Yaskawa INFORM job: OK_R2_O242(-90,180)OKKR.JBI

/JOB
//NAME OK_R2_O242(-90,180)OKKR
///FOLDERNAME X4
//POS
///NPOS 123,123,123,4,0,0
///TOOL 0
///POSTYPE PULSE
///PULSE
C00000=1085,-105763,-105592,1367,57789,-79187
C00001=48587,-61870,-56373,37554,57186,-71211
C00002=109319,-98863,-81663,-17130,36799,-47258
C00003=110499,-70978,-76585,-14581,28064,-55521
C00004=114923,11399,-23396,-32739,57115,-42289
C00005=116623,27529,-9023,-35345,61036,-36673
C00006=106531,29443,-6029,-23966,54360,-54184
C00007=107072,29107,-4870,-24608,53702,-53789
C00008=107072,28853,-4001,-24811,53095,-53633
C00009=107072,28916,-4224,-24758,53250,-53673
C00010=107722,30543,-2610,-25264,53294,-53401
C00011=107072,28916,-4224,-24758,53250,-53673
C00012=111142,26244,-323,-41203,47920,-52388
C00013=110370,28048,1439,-40770,47447,-52585
C00014=111142,26244,-323,-41203,47920,-52388
C00015=118906,20077,-8538,-45056,52999,-50729
C00016=119909,26329,-1133,-46362,52540,-49898
C00017=119909,26168,171,-46853,51920,-49532
C00018=119909,26196,-79,-46760,52037,-49603
C00019=119136,27214,914,-46366,51584,-49791
C00020=119909,26334,-1167,-46350,52555,-49909
C00021=114397,22245,-5862,-42574,50447,-51878
C00022=114678,22860,-3308,-43462,49647,-51288
C00023=115167,24031,-2185,-43822,49818,-51101
C00024=114397,22245,-5862,-42574,50447,-51878
C00025=121530,27687,-2626,-46433,54487,-50098
C00026=123087,41300,13747,-48930,53168,-48397
C00027=123087,41268,14126,-49069,53001,-48291
C00028=123087,41187,15376,-49530,52460,-47945
C00029=123087,41201,15124,-49437,52567,-48015
C00030=122538,42735,16737,-49268,52140,-48077
C00031=123087,41401,12757,-48563,53611,-48677
C00032=122129,71626,35140,-38253,65229,-58469
C00033=121790,71611,37598,-38532,63876,-58094
C00034=121434,69636,35263,-38247,64057,-58328
C00035=122129,71626,35140,-38253,65229,-58469
C00036=120911,36076,-5205,-37468,69020,-59397
C00037=115840,28901,-5746,-41502,62039,-42211
C00038=98316,48041,7032,-8643,64988,-45963
C00039=115260,32848,2305,-42264,59563,-41364
C00040=114901,35009,3238,-41874,59801,-41652
C00041=97501,40962,-317,-1368,65149,-50240
C00042=97537,41051,-224,-1389,65138,-50228
C00043=106513,42706,1459,-20081,69125,-39156
C00044=114834,56426,16290,-34509,77115,-29407
C00045=115518,59095,19228,-34812,77015,-29106
C00046=118968,76239,39289,-36490,75489,-27209
C00047=119068,69741,30113,-36226,77407,-27817
C00048=122206,59988,23685,-43496,73319,-20353
C00049=127814,79238,36559,-32495,95149,-850
C00050=120292,64376,19422,-33176,77212,-56642
C00051=112530,30834,-756,-20739,48722,-51287
C00052=109411,60829,14687,-9556,77735,-26746
C00053=109666,62467,17842,-9701,76678,-26580
C00054=109739,35448,3902,-18618,47607,-52319
C00055=109475,35700,4052,-18391,47587,-52436
C00056=111432,39361,576,-18526,58483,-53933
C00057=120982,47505,9487,-38936,66696,-53604
C00058=124075,44734,17342,-51843,57601,-49295
C00059=126052,54341,27795,-53434,57782,-48179
C00060=126486,54548,28017,-53644,58006,-48066
C00061=128675,70290,46192,-56073,57444,-46208
C00062=128914,63950,33868,-51063,60408,-47630
C00063=125493,46290,11213,-43702,62626,-49802
C00064=121024,34692,-8870,-25769,64212,-48636
C00065=116968,-20453,-45092,-25851,41430,-48067
C00066=118489,-78623,-76964,-34127,32976,-43558
C00067=15896,-74508,-72271,73191,84674,-57421
C00068=31461,-74136,-72097,73237,111249,-57325
C00069=37199,-69408,-69826,73614,107600,-56062
C00070=-3643,-76224,-106676,-19950,71810,-76872
C00071=49550,-101636,-102264,56737,88786,31332
C00072=138514,-74114,-82544,4040,38797,48213
C00073=129498,7065,-37023,9065,67369,37181
C00074=133542,65003,16374,22570,90358,433
C00075=140622,86165,36573,15496,97977,-30873
C00076=140802,90119,43938,15362,95529,-31124
C00077=140802,89712,44636,15338,94910,-31202
C00078=140802,89824,44435,15345,95084,-31180
C00079=141302,92318,47595,15241,94356,-31104
C00080=140802,90328,43607,15371,95825,-31086
C00081=139449,100407,57298,15497,92942,-31904
C00082=140520,104512,63149,15296,91307,-31746
C00083=140782,103254,61503,15262,91612,-31621
C00084=140520,104512,63149,15296,91307,-31746
C00085=139554,101999,57136,15503,93810,-31760
C00086=146528,71128,18474,14629,100276,-28663
C00087=157576,61757,12077,2365,89224,-8186
C00088=158570,72432,22020,167,94145,-8287
C00089=158570,72037,22464,167,93669,-8287
C00090=158570,72148,22336,167,93805,-8287
C00091=157930,73423,23870,319,93520,-8487
C00092=158570,72260,22211,167,93940,-8288
C00093=159049,73117,23241,53,93746,-8137
C00094=159487,76071,26810,-51,93068,-8000
C00095=159049,73117,23241,53,93746,-8137
C00096=152305,60889,6833,1672,97624,-10189
C00097=140378,92804,43752,12660,95661,-26275
C00098=136628,131083,97606,23032,87536,-68506
C00099=138390,134523,104810,22883,84588,-68429
C00100=138286,120316,85504,22190,87431,-66029
C00101=138294,120048,85142,22189,87508,-66012
C00102=139278,110462,71389,17858,93189,-38082
C00103=141573,89787,44718,13729,93335,-28318
C00104=147118,72338,23336,11669,95813,-24471
C00105=147124,72286,23273,11668,95824,-24468
C00106=156033,62541,11743,-1459,94557,-7242
C00107=162183,69089,19251,-9179,95274,2750
C00108=162693,76607,28216,-6950,92750,-113
C00109=162306,74109,24034,-6874,94001,-304
C00110=159278,70446,19892,-6162,94440,-1277
C00111=158953,70496,20103,-6084,94315,-1375
C00112=162506,68092,20237,-10109,87750,-428
C00113=153853,64460,11220,3191,96050,-12949
C00114=153365,70172,19872,3310,93687,-13164
C00115=150414,75792,26653,4027,92524,-14122
C00116=149952,75669,26579,4142,92534,-14265
C00117=143798,90724,45199,9777,90821,-22128
C00118=142426,78831,26541,11541,97051,-24087
C00119=145972,26725,-27800,4713,87219,-24751
C00120=154694,-16289,-62866,-3052,73548,-23707
C00121=178421,-116488,-119781,-18026,60210,-14368
C00122=104141,-125863,-97896,54468,42310,61417
BC00000=193623,514657,895390
BC00001=148789,507467,173552
BC00002=141590,486355,90511
BC00003=133744,463348,17
BC00004=133744,463348,17
BC00005=133744,463348,17
BC00006=133744,463348,17
BC00007=133744,463348,17
BC00008=133744,463348,17
BC00009=133744,463348,17
BC00010=133744,463348,17
BC00011=133744,463348,17
BC00012=133744,463348,17
BC00013=133744,463348,17
BC00014=133744,463348,17
BC00015=133744,463348,17
BC00016=133744,463348,17
BC00017=133744,463348,17
BC00018=133744,463348,17
BC00019=133744,463348,17
BC00020=133744,463348,17
BC00021=133744,463348,17
BC00022=133744,463348,17
BC00023=133744,463348,17
BC00024=133744,463348,17
BC00025=133744,463348,17
BC00026=133744,463348,17
BC00027=133744,463348,17
BC00028=133744,463348,17
BC00029=133744,463348,17
BC00030=133744,463348,17
BC00031=133744,463348,17
BC00032=133744,463348,17
BC00033=133744,463348,17
BC00034=133744,463348,17
BC00035=133744,463348,17
BC00036=133744,463348,17
BC00037=122188,464291,17
BC00038=122188,464291,17
BC00039=122188,464291,17
BC00040=122188,464291,17
BC00041=122188,464291,17
BC00042=122188,464291,17
BC00043=122188,464291,17
BC00044=122188,464291,17
BC00045=122188,464291,17
BC00046=122188,464291,17
BC00047=122188,464291,17
BC00048=122188,464291,17
BC00049=171328,466575,1429
BC00050=151043,472209,15
BC00051=151043,472209,15
BC00052=151042,472210,17
BC00053=151042,472210,17
BC00054=151043,472209,15
BC00055=151043,472209,15
BC00056=151043,472209,15
BC00057=151043,472209,15
BC00058=151043,472209,15
BC00059=151043,472210,15
BC00060=151043,472209,15
BC00061=151043,472209,15
BC00062=151043,472209,15
BC00063=151043,472209,15
BC00064=150303,469416,10754
BC00065=145083,508024,7369
BC00066=145083,506336,7369
BC00067=139738,502478,3904
BC00068=139738,503304,3904
BC00069=139904,513247,3900
BC00070=199448,515539,1075137
BC00071=228950,509401,17
BC00072=305648,462400,17
BC00073=305648,462400,17
BC00074=337500,445626,17
BC00075=364836,431230,17
BC00076=364836,431230,17
BC00077=364836,431230,17
BC00078=364836,431230,17
BC00079=364836,431230,17
BC00080=364836,431230,17
BC00081=364836,431230,17
BC00082=364836,431230,17
BC00083=364836,431230,17
BC00084=364836,431230,17
BC00085=364836,431230,17
BC00086=364836,431230,17
BC00087=364836,431230,17
BC00088=364836,431230,17
BC00089=364836,431230,17
BC00090=364836,431230,17
BC00091=364836,431230,17
BC00092=364836,431230,17
BC00093=364836,431230,17
BC00094=364836,431230,17
BC00095=364836,431230,17
BC00096=364836,431230,17
BC00097=364836,431230,17
BC00098=364836,431230,17
BC00099=364836,431230,17
BC00100=364836,431230,17
BC00101=364836,431230,17
BC00102=364836,431230,17
BC00103=364836,431230,17
BC00104=364836,431230,17
BC00105=364836,431230,17
BC00106=364836,431230,17
BC00107=364836,431230,17
BC00108=364836,431230,17
BC00109=364836,431230,17
BC00110=364836,431230,17
BC00111=364836,431230,17
BC00112=364836,431230,17
BC00113=364836,431230,17
BC00114=364836,431231,13
BC00115=364836,431231,13
BC00116=364836,431231,13
BC00117=364836,431231,13
BC00118=364836,431231,13
BC00119=364836,431231,13
BC00120=364836,431231,13
BC00121=364836,431231,13
BC00122=299887,489577,95909
EC00000=798141,-184050
EC00001=798073,-185062
EC00002=798113,-184473
EC00003=798156,-183832
EC00004=798156,-183832
EC00005=798156,-183832
EC00006=798156,-183832
EC00007=798156,-183832
EC00008=798156,-183832
EC00009=798156,-183832
EC00010=798156,-183832
EC00011=798156,-183832
EC00012=798156,-183832
EC00013=798156,-183832
EC00014=798156,-183832
EC00015=798156,-183832
EC00016=798156,-183832
EC00017=798156,-183832
EC00018=798156,-183832
EC00019=798156,-183832
EC00020=798156,-183832
EC00021=798156,-183832
EC00022=798156,-183832
EC00023=798156,-183832
EC00024=798156,-183832
EC00025=798156,-183832
EC00026=798156,-183832
EC00027=798156,-183832
EC00028=798156,-183832
EC00029=798156,-183832
EC00030=798156,-183832
EC00031=798156,-183832
EC00032=798156,-183832
EC00033=798156,-183832
EC00034=798156,-183832
EC00035=798156,-183832
EC00036=798156,-183832
EC00037=798156,-183832
EC00038=798156,-183832
EC00039=798156,-183832
EC00040=798156,-183832
EC00041=798156,-183832
EC00042=798156,-183832
EC00043=798156,-183832
EC00044=798156,-183832
EC00045=798156,-183832
EC00046=798156,-183832
EC00047=798156,-183832
EC00048=798156,-183832
EC00049=798156,-183832
EC00050=798155,-183832
EC00051=798155,-183832
EC00052=798156,-183832
EC00053=798156,-183832
EC00054=798155,-183832
EC00055=798155,-183832
EC00056=798155,-183832
EC00057=798155,-183832
EC00058=798155,-183832
EC00059=798155,-183832
EC00060=798155,-183832
EC00061=798155,-183832
EC00062=798155,-183832
EC00063=798155,-183832
EC00064=798155,-183832
EC00065=798155,-183832
EC00066=798155,-183832
EC00067=798155,-183832
EC00068=878588,-403504
EC00069=886883,-1018081
EC00070=798156,-1296783
EC00071=798156,-1296783
EC00072=798156,-1296783
EC00073=798156,-1296783
EC00074=798156,-1296783
EC00075=798156,-1296783
EC00076=798156,-1296783
EC00077=798156,-1296783
EC00078=798156,-1296783
EC00079=798156,-1296783
EC00080=798156,-1296783
EC00081=798156,-1296783
EC00082=798156,-1296783
EC00083=798156,-1296783
EC00084=798156,-1296783
EC00085=798156,-1296783
EC00086=798156,-1296783
EC00087=798156,-1296783
EC00088=798156,-1296783
EC00089=798156,-1296783
EC00090=798156,-1296783
EC00091=798156,-1296783
EC00092=798156,-1296783
EC00093=798156,-1296783
EC00094=798156,-1296783
EC00095=798156,-1296783
EC00096=798156,-1296783
EC00097=798156,-1296783
EC00098=798156,-1296783
EC00099=798156,-1296783
EC00100=798156,-1296783
EC00101=798156,-1296783
EC00102=798156,-1296783
EC00103=798156,-1296783
EC00104=798156,-1296783
EC00105=798156,-1296783
EC00106=798156,-1296783
EC00107=798156,-1296783
EC00108=798156,-1296783
EC00109=798156,-1296783
EC00110=798156,-1296783
EC00111=798156,-1296783
EC00112=798156,-1296783
EC00113=798156,-1296783
EC00114=798155,-1296786
EC00115=798155,-1296786
EC00116=798155,-1296786
EC00117=798155,-1296786
EC00118=798155,-1296786
EC00119=798155,-1296786
EC00120=798155,-1296786
EC00121=798155,-1296786
EC00122=798156,-1296783
///POSTYPE BASE
///RECTAN
///RCONF 0,0,0,0,1,0,0,0,0,0,0,0,0,0,0,0,0,0,0,0,0,0,0,0
P00006=2.006,1.622,-0.565,0.0000,0.0000,0.0000
P00021=0.073,2.058,-0.109,0.0000,0.0000,0.0000
P00022=2.006,1.622,-0.565,0.0000,0.0000,0.0000
///RCONF 0,0,0,0,0,0,0,0,0,0,0,0,0,0,0,0,0,0,0,0,0,0,0,0
P00023=-2.957,-4.083,2.762,0.0000,0.0000,0.0000
//INST
///DATE 2024/11/13 18:06
///ATTR SC,RW
///GROUP1 RB1,BS1
///GROUP2 ST1
NOP
'OK_r2_O24.2(-90,180)
'-90,0
MOVJ C00000 BC00000 VJ=100.00  +MOVJ EC00000 VJ=100.00
MOVJ C00001 BC00001 VJ=100.00  +MOVJ EC00001 VJ=25.00
MOVJ C00002 BC00002 VJ=100.00  +MOVJ EC00002 VJ=25.00
MOVJ C00003 BC00003 VJ=100.00  +MOVJ EC00003 VJ=100.00
MOVJ C00004 BC00004 VJ=100.00  +MOVJ EC00004 VJ=25.00
'Path S1574
SFTOF3D
MOVJ C00005 BC00005 VJ=100.00  +MOVJ EC00005 VJ=100.00
MOVL C00006 BC00006 V=166.7  +MOVJ EC00006 VJ=100.00
SMOVL C00007 BC00007 V=100.0  +MOVJ EC00007
SREFP 3 C00008 BC00008  +REFP EC00008
CALL JOB:SEARCH-R1-S13D
SET P021 P006
SFTON3D P021
SMOVL C00009 BC00009 V=100.0  +MOVJ EC00009
SREFP 3 C00010 BC00010  +REFP EC00010
CALL JOB:SEARCH-R1-S13D
SET P021 P006
SFTON3D P021
SMOVL C00011 BC00011 V=100.0  +MOVJ EC00011
SMOVL C00012 BC00012 V=200.0  +MOVJ EC00012
SREFP 3 C00013 BC00013  +REFP EC00013
CALL JOB:SEARCH-R1-S13D
SET P021 P006
SFTON3D P021
SMOVL C00014 BC00014 V=100.0  +MOVJ EC00014
SFTOF3D
MOVL C00015 BC00015 V=400.0  +MOVJ EC00015 VJ=100.00
SMOVL C00016 BC00016 V=133.3  +MOVJ EC00016
SREFP 3 C00017 BC00017  +REFP EC00017
CALL JOB:SEARCH-R1-S13D
SET P022 P006
SFTON3D P022
SMOVL C00018 BC00018 V=100.0  +MOVJ EC00018
SREFP 3 C00019 BC00019  +REFP EC00019
CALL JOB:SEARCH-R1-S13D
SET P022 P006
SFTON3D P022
SMOVL C00020 BC00020 V=100.0  +MOVJ EC00020
SMOVL C00021 BC00021 V=200.0  +MOVJ EC00021
SMOVL C00022 BC00022 V=133.3  +MOVJ EC00022
SREFP 3 C00023 BC00023  +REFP EC00023
CALL JOB:SEARCH-R1-S13D
SET P022 P006
SFTON3D P022
SMOVL C00024 BC00024 V=100.0  +MOVJ EC00024
SFTOF3D
SMOVL C00025 BC00025 V=333.3  +MOVJ EC00025
SMOVL C00026 BC00026 V=166.7  +MOVJ EC00026
SMOVL C00027 BC00027 V=100.0  +MOVJ EC00027
SREFP 3 C00028 BC00028  +REFP EC00028
CALL JOB:SEARCH-R1-S13D
SET P023 P006
SFTON3D P023
SMOVL C00029 BC00029 V=100.0  +MOVJ EC00029
SREFP 3 C00030 BC00030  +REFP EC00030
CALL JOB:SEARCH-R1-S13D
SET P023 P006
SFTON3D P023
SMOVL C00031 BC00031 V=100.0  +MOVJ EC00031
SMOVL C00032 BC00032 V=200.0  +MOVJ EC00032
SMOVL C00033 BC00033 V=166.7  +MOVJ EC00033
SREFP 3 C00034 BC00034  +REFP EC00034
CALL JOB:SEARCH-R1-S13D
SET P023 P006
SFTON3D P023
SMOVL C00035 BC00035 V=200.0  +MOVJ EC00035
SFTOF3D
SMOVL C00036 BC00036 V=500.0  +MOVJ EC00036
'Path W1575
SFTOF3D
SFTON3D P021
MOVJ C00037 BC00037 VJ=100.00  +MOVJ EC00037 VJ=100.00
SMOVL C00038 BC00038 V=166.7 PL=0  +MOVJ EC00038
SREFP 1 C00039 BC00039  +REFP EC00039
SREFP 2 C00040 BC00040  +REFP EC00040
MACRO1 MJ#(0) ARGF9
ARCON
SMOVL C00041 BC00041 V=10.0  +MOVJ EC00041
SMOVC C00042 BC00042 V=10.0  +MOVJ EC00042
SMOVC C00043 BC00043 V=10.0  +MOVJ EC00043
SFTON3D P022
SMOVC C00044 BC00044 V=10.0  +MOVJ EC00044
SMOVC C00045 BC00045 V=10.0  +MOVJ EC00045
SFTON3D P023
SMOVL C00046 BC00046 V=10.0  +MOVJ EC00046
ARCOF
SMOVL C00047 BC00047 V=400.0  +MOVJ EC00047
SMOVL C00048 BC00048 V=1000.0  +MOVJ EC00048
SFTOF3D
'Path W1576
SFTOF3D
SFTON3D P021
SMOVL C00049 BC00049 V=133.3  +MOVJ EC00049
SFTOF3D
SFTON3D P021
SMOVL C00050 BC00050 V=133.3  +MOVJ EC00050
SMOVL C00051 BC00051 V=133.3 PL=0  +MOVJ EC00051
SREFP 1 C00052 BC00052  +REFP EC00052
SREFP 2 C00053 BC00053  +REFP EC00053
MACRO1 MJ#(0) ARGF9
ARCON
SMOVL C00054 BC00054 V=7.5  +MOVJ EC00054
SMOVL C00055 BC00055 V=7.5  +MOVJ EC00055
ARCOF
MOVL C00056 BC00056 V=166.7  +MOVJ EC00056 VJ=25.00
SFTOF3D
MOVL C00057 BC00057 V=250.0  +MOVJ EC00057 VJ=25.00
SFTON3D P022
SMOVL C00058 BC00058 V=133.3  +MOVJ EC00058
ARCON
SMOVL C00059 BC00059 V=7.5  +MOVJ EC00059
SMOVL C00060 BC00060 V=7.5  +MOVJ EC00060
ARCON
SFTON3D P023
SMOVL C00061 BC00061 V=7.5  +MOVJ EC00061
ARCOF
SMOVL C00062 BC00062 V=166.7  +MOVJ EC00062
SMOVL C00063 BC00063 V=400.0  +MOVJ EC00063
SFTOF3D
MOVJ C00064 BC00064 VJ=100.00  +MOVJ EC00064 VJ=100.00
MOVJ C00065 BC00065 VJ=100.00  +MOVJ EC00065 VJ=25.00
MOVJ C00066 BC00066 VJ=100.00  +MOVJ EC00066 VJ=25.00
MOVJ C00067 BC00067 VJ=100.00  +MOVJ EC00067 VJ=100.00
'-90,180
MOVJ C00068 BC00068 VJ=100.00  +MOVJ EC00068 VJ=100.00
MOVJ C00069 BC00069 VJ=100.00  +MOVJ EC00069 VJ=100.00
MOVJ C00070 BC00070 VJ=100.00  +MOVJ EC00070 VJ=100.00
CALL JOB:CLEAN-R1_KM_NEW
MOVJ C00071 BC00071 VJ=100.00  +MOVJ EC00071 VJ=25.00
MOVJ C00072 BC00072 VJ=100.00  +MOVJ EC00072 VJ=100.00
MOVJ C00073 BC00073 VJ=100.00  +MOVJ EC00073 VJ=25.00
'Path S1580
SFTOF3D
MOVJ C00074 BC00074 VJ=100.00  +MOVJ EC00074 VJ=100.00
MOVJ C00075 BC00075 VJ=100.00  +MOVJ EC00075 VJ=100.00
SMOVL C00076 BC00076 V=133.3  +MOVJ EC00076
SREFP 3 C00077 BC00077  +REFP EC00077
CALL JOB:SEARCH-R1-S13D
SET P021 P006
SFTON3D P021
SMOVL C00078 BC00078 V=100.0  +MOVJ EC00078
SREFP 3 C00079 BC00079  +REFP EC00079
CALL JOB:SEARCH-R1-S13D
SET P021 P006
SFTON3D P021
SMOVL C00080 BC00080 V=100.0  +MOVJ EC00080
SMOVL C00081 BC00081 V=166.7  +MOVJ EC00081
SMOVL C00082 BC00082 V=100.0  +MOVJ EC00082
SREFP 3 C00083 BC00083  +REFP EC00083
CALL JOB:SEARCH-R1-S13D
SET P021 P006
SFTON3D P021
SMOVL C00084 BC00084 V=100.0  +MOVJ EC00084
SMOVL C00085 BC00085 V=333.3  +MOVJ EC00085
SFTOF3D
SMOVL C00086 BC00086 V=333.3  +MOVJ EC00086
SMOVL C00087 BC00087 V=333.3  +MOVJ EC00087
SMOVL C00088 BC00088 V=100.0  +MOVJ EC00088
SREFP 3 C00089 BC00089  +REFP EC00089
CALL JOB:SEARCH-R1-S13D
SET P022 P006
SFTON3D P022
SMOVL C00090 BC00090 V=100.0  +MOVJ EC00090
SREFP 3 C00091 BC00091  +REFP EC00091
CALL JOB:SEARCH-R1-S13D
SET P022 P006
SFTON3D P022
SMOVL C00092 BC00092 V=100.0  +MOVJ EC00092
SMOVL C00093 BC00093 V=166.7  +MOVJ EC00093
SREFP 3 C00094 BC00094  +REFP EC00094
CALL JOB:SEARCH-R1-S13D
SET P022 P006
SFTON3D P022
SMOVL C00095 BC00095 V=100.0  +MOVJ EC00095
SFTOF3D
SMOVL C00096 BC00096 V=333.3  +MOVJ EC00096
MOVJ C00097 BC00097 VJ=100.00  +MOVJ EC00097 VJ=100.00
MOVJ C00098 BC00098 VJ=100.00  +MOVJ EC00098 VJ=100.00
MACRO1 MJ#(0) ARGF9
SFTON3D P021
SMOVL C00099 BC00099 V=133.3  +MOVJ EC00099
ARCON
SMOVL C00100 BC00100 V=10.0  +MOVJ EC00100
SMOVC C00101 BC00101 V=10.0  +MOVJ EC00101
SMOVC C00102 BC00102 V=10.0  +MOVJ EC00102
SMOVC C00103 BC00103 V=10.0  +MOVJ EC00103
SMOVL C00104 BC00104 V=10.0  +MOVJ EC00104
SMOVC C00105 BC00105 V=10.0  +MOVJ EC00105
SFTON3D P022
SMOVC C00106 BC00106 V=10.0  +MOVJ EC00106
SMOVC C00107 BC00107 V=10.0  +MOVJ EC00107
SMOVL C00108 BC00108 V=10.0  +MOVJ EC00108
ARCOF
SMOVL C00109 BC00109 V=166.7  +MOVJ EC00109
SFTOF3D
SMOVL C00110 BC00110 V=166.7  +MOVJ EC00110
SFTON3D P022
SMOVL C00111 BC00111 V=166.7  +MOVJ EC00111
ARCON
SMOVL C00112 BC00112 V=8.3  +MOVJ EC00112
ARCOF
SFTOF3D
SMOVL C00113 BC00113 V=166.7  +MOVJ EC00113
SFTON3D P021
SMOVL C00114 BC00114 V=10.0  +MOVJ EC00114
ARCON
SMOVL C00115 BC00115 V=8.3  +MOVJ EC00115
SMOVL C00116 BC00116 V=8.3  +MOVJ EC00116
SMOVL C00117 BC00117 V=8.3  +MOVJ EC00117
ARCOF
SMOVL C00118 BC00118 V=333.3  +MOVJ EC00118
SFTOF3D
MOVJ C00119 BC00119 VJ=100.00  +MOVJ EC00119 VJ=100.00
MOVJ C00120 BC00120 VJ=100.00  +MOVJ EC00120 VJ=100.00
MOVJ C00121 BC00121 VJ=100.00  +MOVJ EC00121 VJ=100.00
SFTOF3D
MOVJ C00122 BC00122 VJ=100.00  +MOVJ EC00122 VJ=100.00
END
